# EPICS substitutions: ek9000App/Db/EL3141.substitutions
file EL3141.template
{       pattern
        {
                TERMINAL,

        }
        {
        }
}
